// TIA Portal V20 export
DATA_BLOCK "DB_GestionFixture"   // DB89
// stored: InstanceOfName FB_GestionFixture, InstanceOfType FB
"FB_GestionFixture"
   // VAR RETAIN
   //    sFixtureHold : Bool;
   // END_VAR
   // VAR
   //    sFixtureVacuum : Bool;
   //    sFixtureBlowing : Bool;
   //    sFixtureStandard { S7_SetPoint := 'True'} : "FB_Fixture";
   //    sFixtureStandardErrorCode { S7_SetPoint := 'True'} : Int;
   //    sFixturePartControl : "FB_PartPresenceCtrl";
   //    sRT_VacuumStartReq { S7_SetPoint := 'True'} : R_TRIG;
   //    sRT_VacuumStopReq { S7_SetPoint := 'True'} : R_TRIG;
   // END_VAR
BEGIN
END_DATA_BLOCK
